PROGRAM EM01_Robot
VAR
	
	//Backbone
	FB_StateMachine_Robot			: FB_StateManager;
	bFl_RunningMachineRobot			: BOOL;
	bFl_SeqReset					: BOOL;
	Bypass_Safety					: BOOL;
	bFl_Manual						: BOOL;
	CheckStatusRobot				: checkstatus;
	AlarmEventHistory				: ARRAY[1..20] OF Alarm_Event_History;
	StartUpRobot					: FB_StartUpRobot;
	AlarmEventActive				: ARRAY[1..20] OF Alarm_Event_Active;
	Connection_Robot				: TON;
END_VAR
VAR // added by the converter: edge detectors and wires of the graphical bodies
    _w1, _w2, _w3, _w4 : BOOL;
END_VAR

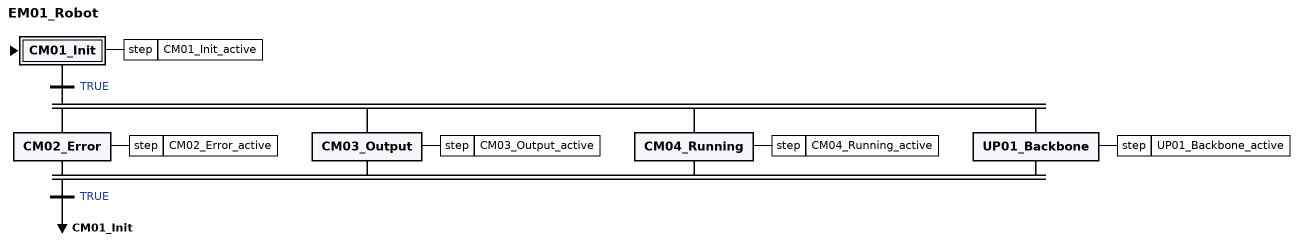
INITIAL_STEP CM01_Init:
    CM01_Init_active(N);  // step action
END_STEP
TRANSITION FROM CM01_Init TO (CM02_Error, CM03_Output, CM04_Running, UP01_Backbone)
    := TRUE;
END_TRANSITION
STEP CM02_Error:
    CM02_Error_active(N);  // step action
END_STEP
STEP CM03_Output:
    CM03_Output_active(N);  // step action
END_STEP
STEP CM04_Running:
    CM04_Running_active(N);  // step action
END_STEP
STEP UP01_Backbone:
    UP01_Backbone_active(N);  // step action
END_STEP
TRANSITION FROM (CM02_Error, CM03_Output, CM04_Running, UP01_Backbone) TO CM01_Init
    := TRUE;
END_TRANSITION

ACTION CM01_Init_active:
Data_GVL.bFL_StartRobot				:= Status_GVL.bFl_RunButton_Robotic OR HMI_GVL.bStartButtonRobot;
Data_GVL.bFL_StopRobot				:= NOT Status_GVL.bFl_StopButton_Robotic OR HMI_GVL.bStopButtonRobot;
Data_GVL.bFL_ResetRobot				:= Status_GVL.bFl_ResetButton_Robotic OR HMI_GVL.bResetButtonRobot;
Data_GVL.bFL_AckRobot				:= Status_GVL.bFl_Acknowledge_Robotic OR HMI_GVL.bAcknowledgeButtonRobot;
Data_GVL.bFL_AutoManuaModeRobot 	:= Status_GVL.bFl_Manual_Robotic OR HMI_GVL.bTestModeEnableRobot;
bFl_RunningMachineRobot				:= Data_GVL.stStateMachineRobot.Running;
bFl_Manual							:= Data_GVL.stStateMachineRobot.ManualMode;
bFl_SeqReset						:= NOT Status_GVL.bFl_EStop_Robotic OR InputOutput_GVL.xIn_Robot.StsSupervision OR InputOutput_GVL.xIn_Robot.StsEmergencyStop OR NOT InputOutput_GVL.xIn_Robot.StsAutoOn;



(*=================Convert Timer============================*)
END_ACTION

ACTION CM02_Error_active:
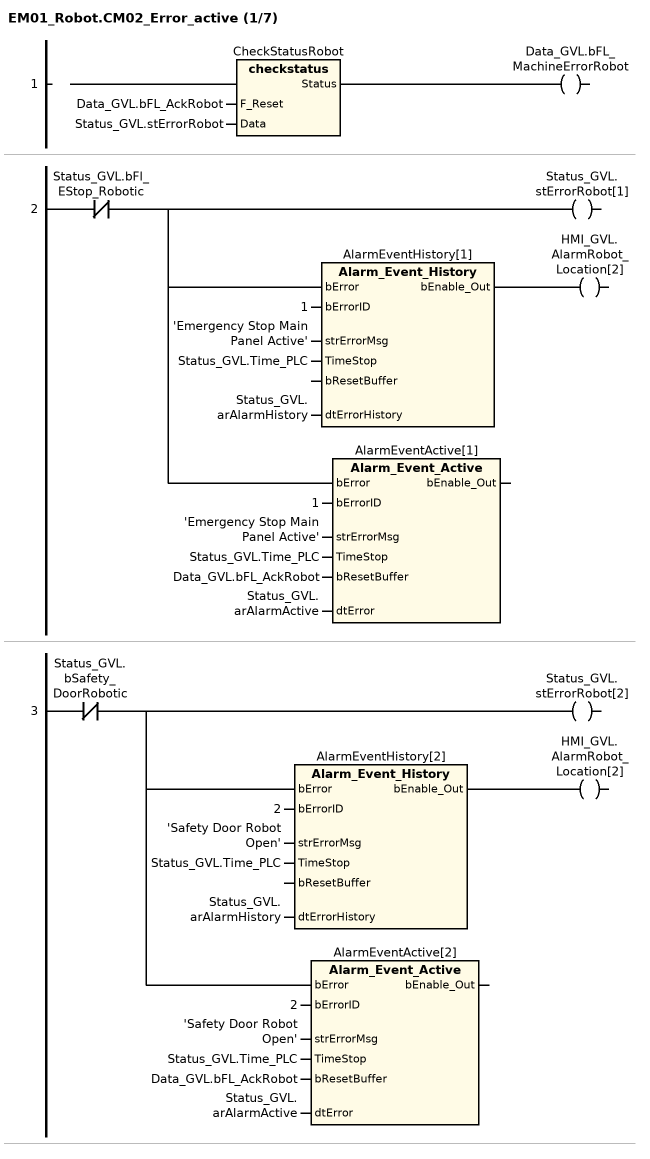
// NETWORK 1
CheckStatusRobot(F_Reset := Data_GVL.bFL_AckRobot, Data := Status_GVL.stErrorRobot); // checkstatus
Data_GVL.bFL_MachineErrorRobot := CheckStatusRobot.Status;

// NETWORK 2
_w1 := NOT Status_GVL.bFl_EStop_Robotic;
Status_GVL.stErrorRobot[1] := _w1;
AlarmEventHistory[1](
    bError := _w1,
    bErrorID := 1,
    strErrorMsg := 'Emergency Stop Main Panel Active',
    TimeStop := Status_GVL.Time_PLC,
    dtErrorHistory := Status_GVL.arAlarmHistory); // Alarm_Event_History
HMI_GVL.AlarmRobot_Location[2] := AlarmEventHistory[1].bEnable_Out;
AlarmEventActive[1](
    bError := _w1,
    bErrorID := 1,
    strErrorMsg := 'Emergency Stop Main Panel Active',
    TimeStop := Status_GVL.Time_PLC,
    bResetBuffer := Data_GVL.bFL_AckRobot,
    dtError := Status_GVL.arAlarmActive); // Alarm_Event_Active

// NETWORK 3
_w2 := NOT Status_GVL.bSafety_DoorRobotic;
Status_GVL.stErrorRobot[2] := _w2;
AlarmEventHistory[2](
    bError := _w2,
    bErrorID := 2,
    strErrorMsg := 'Safety Door Robot Open',
    TimeStop := Status_GVL.Time_PLC,
    dtErrorHistory := Status_GVL.arAlarmHistory); // Alarm_Event_History
HMI_GVL.AlarmRobot_Location[2] := AlarmEventHistory[2].bEnable_Out;
AlarmEventActive[2](
    bError := _w2,
    bErrorID := 2,
    strErrorMsg := 'Safety Door Robot Open',
    TimeStop := Status_GVL.Time_PLC,
    bResetBuffer := Data_GVL.bFL_AckRobot,
    dtError := Status_GVL.arAlarmActive); // Alarm_Event_Active

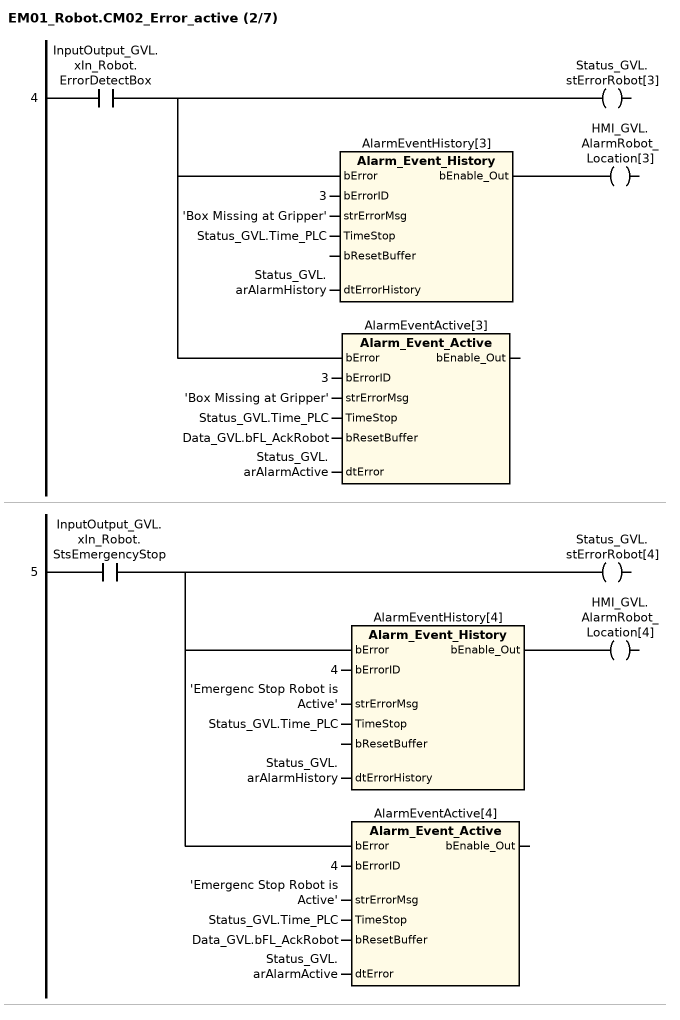
// NETWORK 4
Status_GVL.stErrorRobot[3] := InputOutput_GVL.xIn_Robot.ErrorDetectBox;
AlarmEventHistory[3](
    bError := InputOutput_GVL.xIn_Robot.ErrorDetectBox,
    bErrorID := 3,
    strErrorMsg := 'Box Missing at Gripper',
    TimeStop := Status_GVL.Time_PLC,
    dtErrorHistory := Status_GVL.arAlarmHistory); // Alarm_Event_History
HMI_GVL.AlarmRobot_Location[3] := AlarmEventHistory[3].bEnable_Out;
AlarmEventActive[3](
    bError := InputOutput_GVL.xIn_Robot.ErrorDetectBox,
    bErrorID := 3,
    strErrorMsg := 'Box Missing at Gripper',
    TimeStop := Status_GVL.Time_PLC,
    bResetBuffer := Data_GVL.bFL_AckRobot,
    dtError := Status_GVL.arAlarmActive); // Alarm_Event_Active

// NETWORK 5
Status_GVL.stErrorRobot[4] := InputOutput_GVL.xIn_Robot.StsEmergencyStop;
AlarmEventHistory[4](
    bError := InputOutput_GVL.xIn_Robot.StsEmergencyStop,
    bErrorID := 4,
    strErrorMsg := 'Emergenc Stop Robot is Active',
    TimeStop := Status_GVL.Time_PLC,
    dtErrorHistory := Status_GVL.arAlarmHistory); // Alarm_Event_History
HMI_GVL.AlarmRobot_Location[4] := AlarmEventHistory[4].bEnable_Out;
AlarmEventActive[4](
    bError := InputOutput_GVL.xIn_Robot.StsEmergencyStop,
    bErrorID := 4,
    strErrorMsg := 'Emergenc Stop Robot is Active',
    TimeStop := Status_GVL.Time_PLC,
    bResetBuffer := Data_GVL.bFL_AckRobot,
    dtError := Status_GVL.arAlarmActive); // Alarm_Event_Active

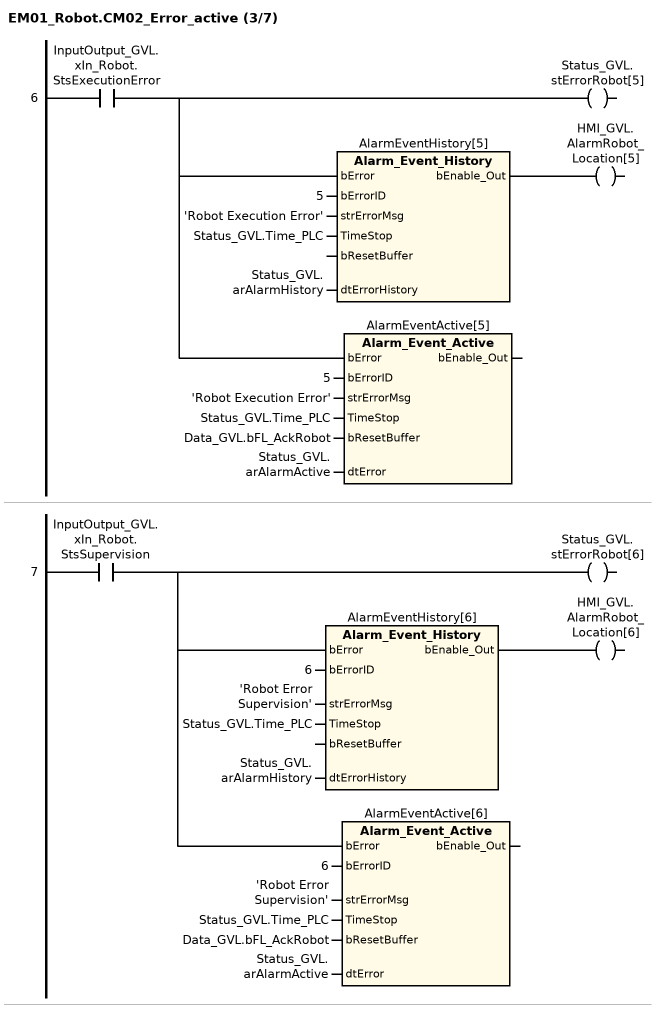
// NETWORK 6
Status_GVL.stErrorRobot[5] := InputOutput_GVL.xIn_Robot.StsExecutionError;
AlarmEventHistory[5](
    bError := InputOutput_GVL.xIn_Robot.StsExecutionError,
    bErrorID := 5,
    strErrorMsg := 'Robot Execution Error',
    TimeStop := Status_GVL.Time_PLC,
    dtErrorHistory := Status_GVL.arAlarmHistory); // Alarm_Event_History
HMI_GVL.AlarmRobot_Location[5] := AlarmEventHistory[5].bEnable_Out;
AlarmEventActive[5](
    bError := InputOutput_GVL.xIn_Robot.StsExecutionError,
    bErrorID := 5,
    strErrorMsg := 'Robot Execution Error',
    TimeStop := Status_GVL.Time_PLC,
    bResetBuffer := Data_GVL.bFL_AckRobot,
    dtError := Status_GVL.arAlarmActive); // Alarm_Event_Active

// NETWORK 7
Status_GVL.stErrorRobot[6] := InputOutput_GVL.xIn_Robot.StsSupervision;
AlarmEventHistory[6](
    bError := InputOutput_GVL.xIn_Robot.StsSupervision,
    bErrorID := 6,
    strErrorMsg := 'Robot Error Supervision',
    TimeStop := Status_GVL.Time_PLC,
    dtErrorHistory := Status_GVL.arAlarmHistory); // Alarm_Event_History
HMI_GVL.AlarmRobot_Location[6] := AlarmEventHistory[6].bEnable_Out;
AlarmEventActive[6](
    bError := InputOutput_GVL.xIn_Robot.StsSupervision,
    bErrorID := 6,
    strErrorMsg := 'Robot Error Supervision',
    TimeStop := Status_GVL.Time_PLC,
    bResetBuffer := Data_GVL.bFL_AckRobot,
    dtError := Status_GVL.arAlarmActive); // Alarm_Event_Active

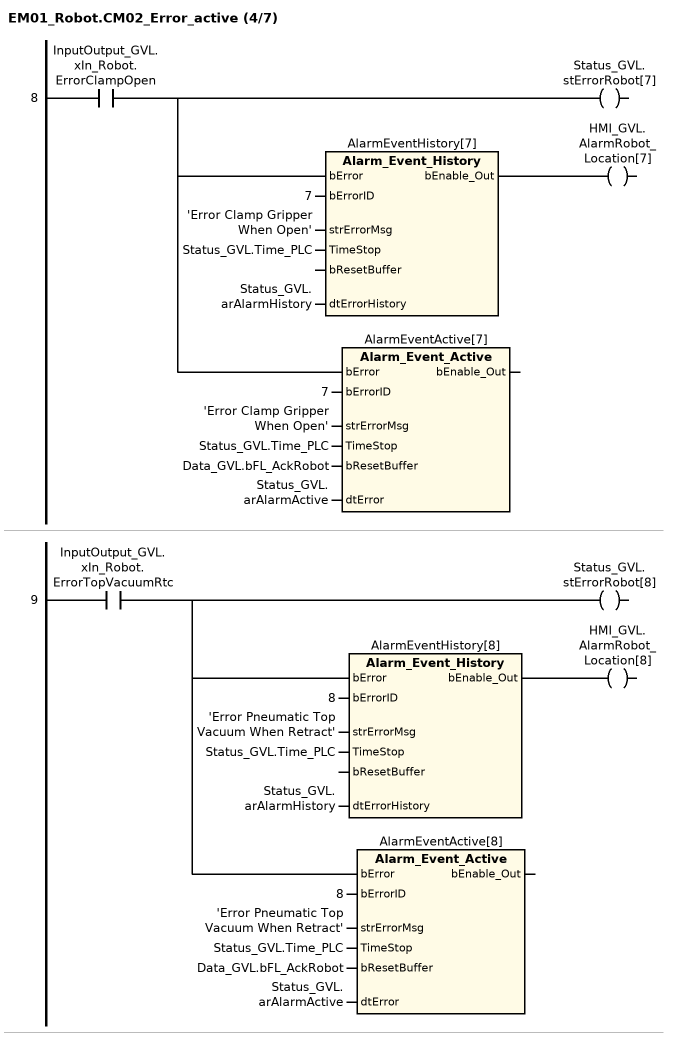
// NETWORK 8
Status_GVL.stErrorRobot[7] := InputOutput_GVL.xIn_Robot.ErrorClampOpen;
AlarmEventHistory[7](
    bError := InputOutput_GVL.xIn_Robot.ErrorClampOpen,
    bErrorID := 7,
    strErrorMsg := 'Error Clamp Gripper When Open',
    TimeStop := Status_GVL.Time_PLC,
    dtErrorHistory := Status_GVL.arAlarmHistory); // Alarm_Event_History
HMI_GVL.AlarmRobot_Location[7] := AlarmEventHistory[7].bEnable_Out;
AlarmEventActive[7](
    bError := InputOutput_GVL.xIn_Robot.ErrorClampOpen,
    bErrorID := 7,
    strErrorMsg := 'Error Clamp Gripper When Open',
    TimeStop := Status_GVL.Time_PLC,
    bResetBuffer := Data_GVL.bFL_AckRobot,
    dtError := Status_GVL.arAlarmActive); // Alarm_Event_Active

// NETWORK 9
Status_GVL.stErrorRobot[8] := InputOutput_GVL.xIn_Robot.ErrorTopVacuumRtc;
AlarmEventHistory[8](
    bError := InputOutput_GVL.xIn_Robot.ErrorTopVacuumRtc,
    bErrorID := 8,
    strErrorMsg := 'Error Pneumatic Top Vacuum When Retract',
    TimeStop := Status_GVL.Time_PLC,
    dtErrorHistory := Status_GVL.arAlarmHistory); // Alarm_Event_History
HMI_GVL.AlarmRobot_Location[8] := AlarmEventHistory[8].bEnable_Out;
AlarmEventActive[8](
    bError := InputOutput_GVL.xIn_Robot.ErrorTopVacuumRtc,
    bErrorID := 8,
    strErrorMsg := 'Error Pneumatic Top Vacuum When Retract',
    TimeStop := Status_GVL.Time_PLC,
    bResetBuffer := Data_GVL.bFL_AckRobot,
    dtError := Status_GVL.arAlarmActive); // Alarm_Event_Active

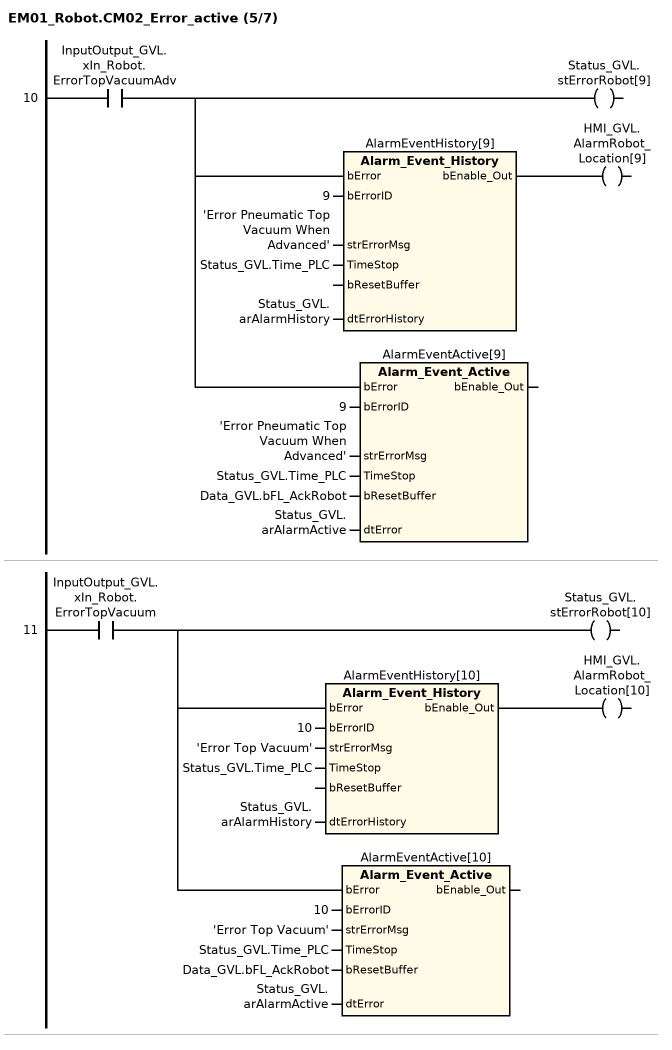
// NETWORK 10
Status_GVL.stErrorRobot[9] := InputOutput_GVL.xIn_Robot.ErrorTopVacuumAdv;
AlarmEventHistory[9](
    bError := InputOutput_GVL.xIn_Robot.ErrorTopVacuumAdv,
    bErrorID := 9,
    strErrorMsg := 'Error Pneumatic Top Vacuum When Advanced',
    TimeStop := Status_GVL.Time_PLC,
    dtErrorHistory := Status_GVL.arAlarmHistory); // Alarm_Event_History
HMI_GVL.AlarmRobot_Location[9] := AlarmEventHistory[9].bEnable_Out;
AlarmEventActive[9](
    bError := InputOutput_GVL.xIn_Robot.ErrorTopVacuumAdv,
    bErrorID := 9,
    strErrorMsg := 'Error Pneumatic Top Vacuum When Advanced',
    TimeStop := Status_GVL.Time_PLC,
    bResetBuffer := Data_GVL.bFL_AckRobot,
    dtError := Status_GVL.arAlarmActive); // Alarm_Event_Active

// NETWORK 11
Status_GVL.stErrorRobot[10] := InputOutput_GVL.xIn_Robot.ErrorTopVacuum;
AlarmEventHistory[10](
    bError := InputOutput_GVL.xIn_Robot.ErrorTopVacuum,
    bErrorID := 10,
    strErrorMsg := 'Error Top Vacuum',
    TimeStop := Status_GVL.Time_PLC,
    dtErrorHistory := Status_GVL.arAlarmHistory); // Alarm_Event_History
HMI_GVL.AlarmRobot_Location[10] := AlarmEventHistory[10].bEnable_Out;
AlarmEventActive[10](
    bError := InputOutput_GVL.xIn_Robot.ErrorTopVacuum,
    bErrorID := 10,
    strErrorMsg := 'Error Top Vacuum',
    TimeStop := Status_GVL.Time_PLC,
    bResetBuffer := Data_GVL.bFL_AckRobot,
    dtError := Status_GVL.arAlarmActive); // Alarm_Event_Active

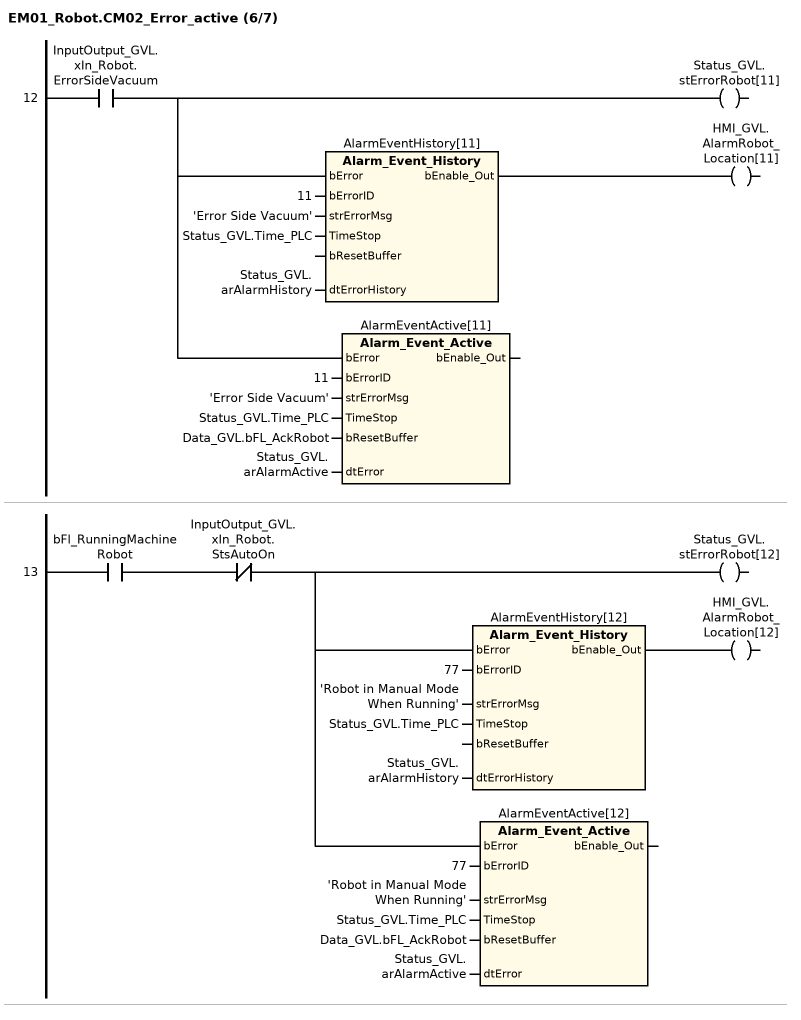
// NETWORK 12
Status_GVL.stErrorRobot[11] := InputOutput_GVL.xIn_Robot.ErrorSideVacuum;
AlarmEventHistory[11](
    bError := InputOutput_GVL.xIn_Robot.ErrorSideVacuum,
    bErrorID := 11,
    strErrorMsg := 'Error Side Vacuum',
    TimeStop := Status_GVL.Time_PLC,
    dtErrorHistory := Status_GVL.arAlarmHistory); // Alarm_Event_History
HMI_GVL.AlarmRobot_Location[11] := AlarmEventHistory[11].bEnable_Out;
AlarmEventActive[11](
    bError := InputOutput_GVL.xIn_Robot.ErrorSideVacuum,
    bErrorID := 11,
    strErrorMsg := 'Error Side Vacuum',
    TimeStop := Status_GVL.Time_PLC,
    bResetBuffer := Data_GVL.bFL_AckRobot,
    dtError := Status_GVL.arAlarmActive); // Alarm_Event_Active

// NETWORK 13
_w3 := bFl_RunningMachineRobot AND NOT InputOutput_GVL.xIn_Robot.StsAutoOn;
Status_GVL.stErrorRobot[12] := _w3;
AlarmEventHistory[12](
    bError := _w3,
    bErrorID := 77,
    strErrorMsg := 'Robot in Manual Mode When Running',
    TimeStop := Status_GVL.Time_PLC,
    dtErrorHistory := Status_GVL.arAlarmHistory); // Alarm_Event_History
HMI_GVL.AlarmRobot_Location[12] := AlarmEventHistory[12].bEnable_Out;
AlarmEventActive[12](
    bError := _w3,
    bErrorID := 77,
    strErrorMsg := 'Robot in Manual Mode When Running',
    TimeStop := Status_GVL.Time_PLC,
    bResetBuffer := Data_GVL.bFL_AckRobot,
    dtError := Status_GVL.arAlarmActive); // Alarm_Event_Active

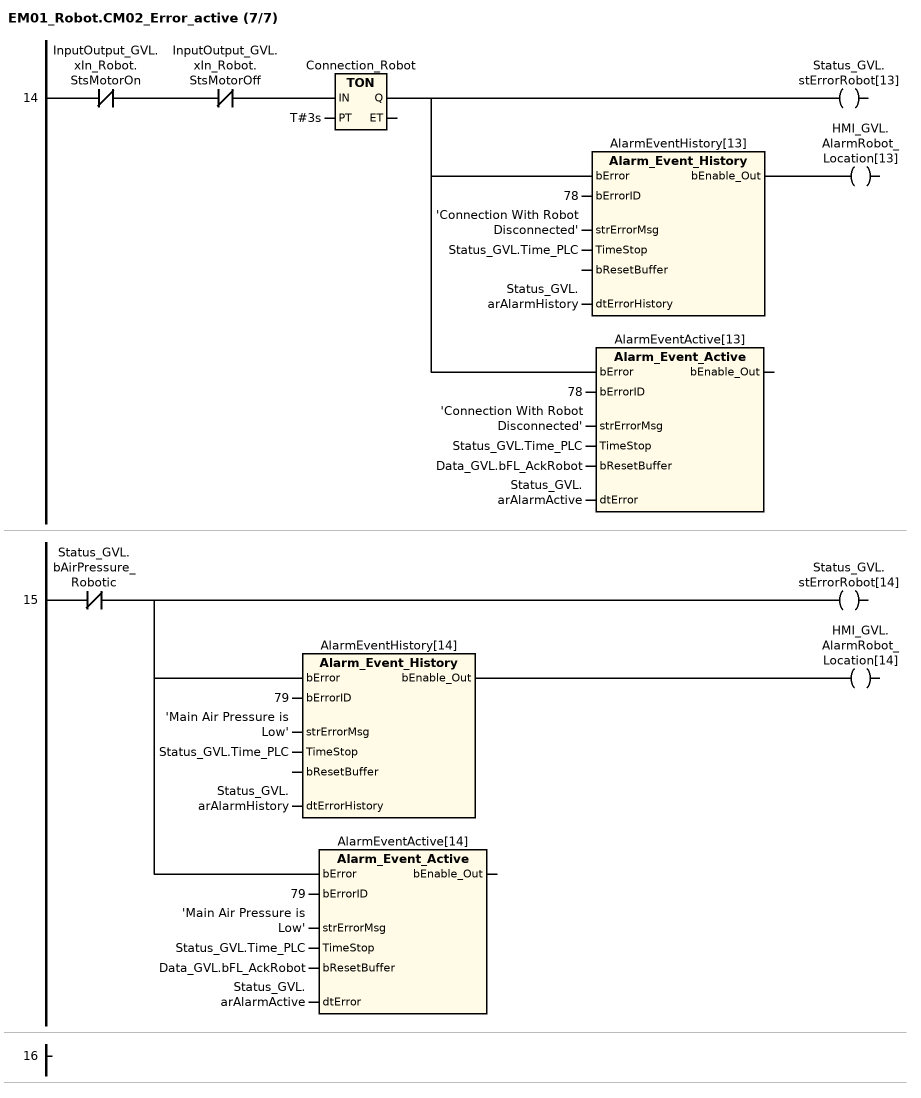
// NETWORK 14
Connection_Robot(IN := NOT InputOutput_GVL.xIn_Robot.StsMotorOn AND NOT InputOutput_GVL.xIn_Robot.StsMotorOff, PT := T#3s); // TON
Status_GVL.stErrorRobot[13] := Connection_Robot.Q;
AlarmEventHistory[13](
    bError := Connection_Robot.Q,
    bErrorID := 78,
    strErrorMsg := 'Connection With Robot Disconnected',
    TimeStop := Status_GVL.Time_PLC,
    dtErrorHistory := Status_GVL.arAlarmHistory); // Alarm_Event_History
HMI_GVL.AlarmRobot_Location[13] := AlarmEventHistory[13].bEnable_Out;
AlarmEventActive[13](
    bError := Connection_Robot.Q,
    bErrorID := 78,
    strErrorMsg := 'Connection With Robot Disconnected',
    TimeStop := Status_GVL.Time_PLC,
    bResetBuffer := Data_GVL.bFL_AckRobot,
    dtError := Status_GVL.arAlarmActive); // Alarm_Event_Active

// NETWORK 15
_w4 := NOT Status_GVL.bAirPressure_Robotic;
Status_GVL.stErrorRobot[14] := _w4;
AlarmEventHistory[14](
    bError := _w4,
    bErrorID := 79,
    strErrorMsg := 'Main Air Pressure is Low',
    TimeStop := Status_GVL.Time_PLC,
    dtErrorHistory := Status_GVL.arAlarmHistory); // Alarm_Event_History
HMI_GVL.AlarmRobot_Location[14] := AlarmEventHistory[14].bEnable_Out;
AlarmEventActive[14](
    bError := _w4,
    bErrorID := 79,
    strErrorMsg := 'Main Air Pressure is Low',
    TimeStop := Status_GVL.Time_PLC,
    bResetBuffer := Data_GVL.bFL_AckRobot,
    dtError := Status_GVL.arAlarmActive); // Alarm_Event_Active

// NETWORK 16
END_ACTION

ACTION CM03_Output_active:
// NETWORK 1 (disabled)
// label: Output Robot
END_ACTION

ACTION CM04_Running_active:
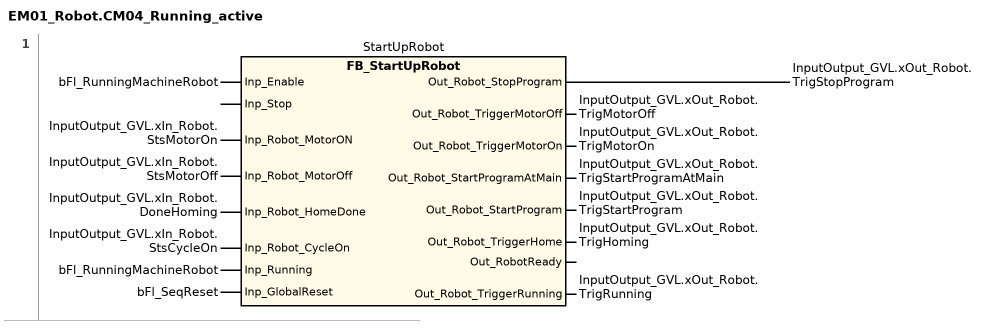
// NETWORK 1
StartUpRobot(
    Inp_Enable := bFl_RunningMachineRobot,
    Inp_Robot_MotorON := InputOutput_GVL.xIn_Robot.StsMotorOn,
    Inp_Robot_MotorOff := InputOutput_GVL.xIn_Robot.StsMotorOff,
    Inp_Robot_HomeDone := InputOutput_GVL.xIn_Robot.DoneHoming,
    Inp_Robot_CycleOn := InputOutput_GVL.xIn_Robot.StsCycleOn,
    Inp_Running := bFl_RunningMachineRobot,
    Inp_GlobalReset := bFl_SeqReset,
    Out_Robot_TriggerMotorOff => InputOutput_GVL.xOut_Robot.TrigMotorOff,
    Out_Robot_TriggerMotorOn => InputOutput_GVL.xOut_Robot.TrigMotorOn,
    Out_Robot_StartProgramAtMain => InputOutput_GVL.xOut_Robot.TrigStartProgramAtMain,
    Out_Robot_StartProgram => InputOutput_GVL.xOut_Robot.TrigStartProgram,
    Out_Robot_TriggerHome => InputOutput_GVL.xOut_Robot.TrigHoming,
    Out_Robot_TriggerRunning => InputOutput_GVL.xOut_Robot.TrigRunning); // FB_StartUpRobot
InputOutput_GVL.xOut_Robot.TrigStopProgram := StartUpRobot.Out_Robot_StopProgram;
END_ACTION

ACTION UP01_Backbone_active:
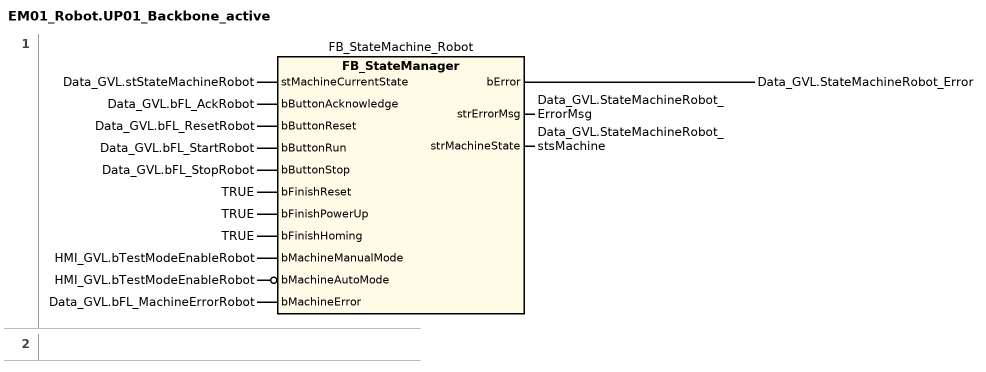
// NETWORK 1
FB_StateMachine_Robot(
    stMachineCurrentState := Data_GVL.stStateMachineRobot,
    bButtonAcknowledge := Data_GVL.bFL_AckRobot,
    bButtonReset := Data_GVL.bFL_ResetRobot,
    bButtonRun := Data_GVL.bFL_StartRobot,
    bButtonStop := Data_GVL.bFL_StopRobot,
    bFinishReset := TRUE,
    bFinishPowerUp := TRUE,
    bFinishHoming := TRUE,
    bMachineManualMode := HMI_GVL.bTestModeEnableRobot,
    bMachineAutoMode := NOT HMI_GVL.bTestModeEnableRobot,
    bMachineError := Data_GVL.bFL_MachineErrorRobot,
    strErrorMsg => Data_GVL.StateMachineRobot_ErrorMsg,
    strMachineState => Data_GVL.StateMachineRobot_stsMachine); // FB_StateManager
Data_GVL.StateMachineRobot_Error := FB_StateMachine_Robot.bError;

// NETWORK 2
END_ACTION

END_PROGRAM

(* stored: Version 1.1.0.1, ProductVersion 3.1.4024.12
   POU EM01_Robot: Id {9ad730f6-91ca-432c-b857-de5fa7db9f33}, SpecialFunc None
   Action CM01_Init_active: Id {6b152d4d-908d-4720-bca8-fd6a24839c6d}
   Action CM02_Error_active: Id {ffeb5f13-b424-4403-ac96-f4cb5076e24a}
   Action CM03_Output_active: Id {67ad0336-c05f-4b1d-adb8-0633041a49d0}
   Action CM04_Running_active: Id {453e4bab-be63-4431-bd62-06895309973c}
   Action UP01_Backbone_active: Id {ef90070c-25e3-41c2-8495-4d0b1b3c399a} *)
